// TIA Portal V16 export
// export: Created 2021-08-30T10:49:31.2193227Z, ExportSetting WithDefaults, DisplayName Totally Integrated Automation Portal, DisplayVersion V16 Update 3, DisplayName TIA Portal Version Control Interface, DisplayVersion V16 Update 2, DisplayName TIA Portal Openness, DisplayVersion V16 Update 3, DisplayName TIA Portal Teamcenter Gateway, DisplayVersion V16, DisplayName STEP 7 Professional, DisplayVersion V16 Update 3, DisplayName STEP 7 Safety, DisplayVersion V16, DisplayName WinCC Advanced, DisplayVersion V16 Update 3
FUNCTION_BLOCK "AvAckAlarm"   // FB48, LAD
{ S7_Optimized_Access := 'TRUE' }
VERSION : 0.1
// stored: AutoNumber true, IsIECCheckEnabled false, IsRetainMemResEnabled false, MemoryReserve 100, SetENOAutomatically false, UDAEnableTagReadback false
   VAR_INPUT
      ack : Bool;
      power : Bool;
      alarmFC : Bool;
      emrStop : Bool;   // Авариный стоп 0-авария, 1-ок
      local : Bool;   // 1-местный режим
      tmrOpening_Q : Bool;
      tmrClosing_Q : Bool;
   END_VAR
   VAR_IN_OUT
      dev : "Av";
      errService : Bool;
      ErrPower : Bool;   // Признак аварии питания
      errAlarmFc : Bool;
      ErrDis : Bool;   // Признак внешней блокировки
      errEmrStop : Bool;
      errLocal : Bool;
      errStart : Bool;
      errStop : Bool;
   END_VAR
   VAR
      InstService { S7_SetPoint := 'True'} : "DevAckSingleAlarm";
      InstPower { S7_SetPoint := 'True'} : "DevAckSingleAlarm";
      InstFc { S7_SetPoint := 'True'} : "DevAckSingleAlarm";
      InstDis { S7_SetPoint := 'True'} : "DevBlockAckSingleAlarm";
      InstEmrStop { S7_SetPoint := 'True'} : "DevAckSingleAlarm";
      InstLocal { S7_SetPoint := 'True'} : "DevAckSingleAlarm";
      InstStart { S7_SetPoint := 'True'} : "DevAckSingleAlarm";
      InstStop { S7_SetPoint := 'True'} : "DevAckSingleAlarm";
   END_VAR
BEGIN

REGION Network 1: Ошибка питания - нужно квитирование ACK
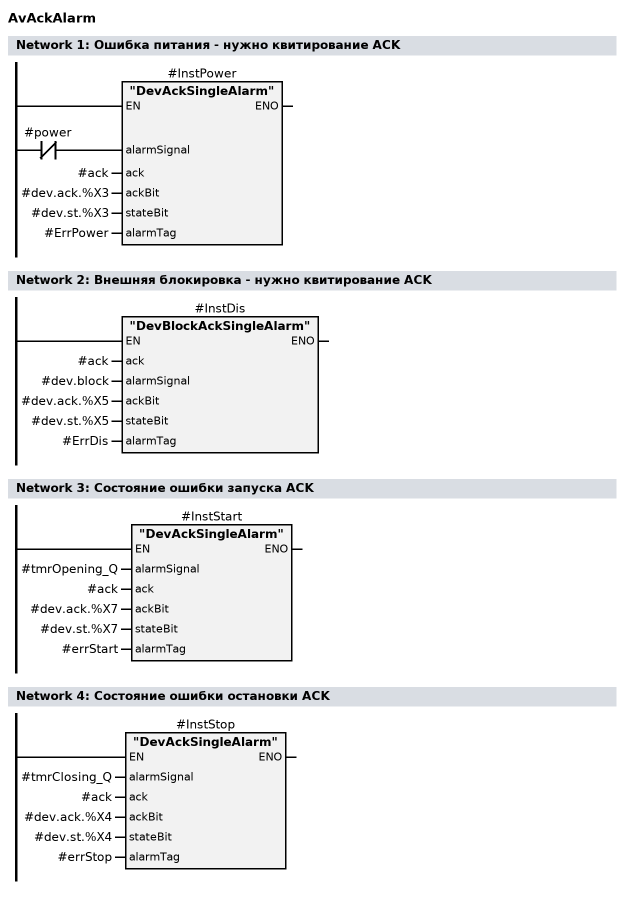
   RUNG wire#powerrail
      #InstPower(alarmSignal := wire#w1, ack := #ack, ackBit := #dev.ack.%X3, stateBit := #dev.st.%X3, alarmTag := #ErrPower)
   END_RUNG
   RUNG wire#powerrail
      I_Contact( #power )
   END_RUNG wire#w1
   // the same network as SCL:
   #InstPower(alarmSignal := NOT #power,   // "DevAckSingleAlarm"
              ack := #ack,
              ackBit := #dev.ack.%X3,
              stateBit := #dev.st.%X3,
              alarmTag := #ErrPower);
END_REGION

REGION Network 2: Внешняя блокировка - нужно квитирование ACK
   RUNG wire#powerrail
      #InstDis(ack := #ack, alarmSignal := #dev.block, ackBit := #dev.ack.%X5, stateBit := #dev.st.%X5, alarmTag := #ErrDis)
   END_RUNG
   // the same network as SCL:
   #InstDis(ack := #ack,   // "DevBlockAckSingleAlarm"
            alarmSignal := #dev.block,
            ackBit := #dev.ack.%X5,
            stateBit := #dev.st.%X5,
            alarmTag := #ErrDis);
END_REGION

REGION Network 3: Состояние ошибки запуска ACK
   RUNG wire#powerrail
      #InstStart(alarmSignal := #tmrOpening_Q, ack := #ack, ackBit := #dev.ack.%X7, stateBit := #dev.st.%X7, alarmTag := #errStart)
   END_RUNG
   // the same network as SCL:
   #InstStart(alarmSignal := #tmrOpening_Q,   // "DevAckSingleAlarm"
              ack := #ack,
              ackBit := #dev.ack.%X7,
              stateBit := #dev.st.%X7,
              alarmTag := #errStart);
END_REGION

REGION Network 4: Состояние ошибки остановки ACK
   RUNG wire#powerrail
      #InstStop(alarmSignal := #tmrClosing_Q, ack := #ack, ackBit := #dev.ack.%X4, stateBit := #dev.st.%X4, alarmTag := #errStop)
   END_RUNG
   // the same network as SCL:
   #InstStop(alarmSignal := #tmrClosing_Q,   // "DevAckSingleAlarm"
             ack := #ack,
             ackBit := #dev.ack.%X4,
             stateBit := #dev.st.%X4,
             alarmTag := #errStop);
END_REGION
END_FUNCTION_BLOCK
